// TIA Portal V20 export
// export: Created 2025-12-01T14:57:05.1586279Z, ExportSetting None, DisplayName Totally Integrated Automation Portal, DisplayVersion V20 Update 3, DisplayName TIA Portal Openness, DisplayVersion V20 Update 3, DisplayName TIA Portal Version Control Interface, DisplayVersion V20 Update 3, DisplayName STEP 7 Professional, DisplayVersion V20 Update 3, DisplayName STEP 7 Safety, DisplayVersion V20 Update 2, DisplayName WinCC Basic/Comfort/Advanced, DisplayVersion V20 Update 3, DisplayName WinCC Professional, DisplayVersion V20 Update 3, DisplayName WinCC Unified, DisplayVersion V20 Update 3
FUNCTION "FC806_JDT01Borrado" : Void   // FC806, LAD
TITLE = "BorrodoTracking" - Borrado de toda la Base de Datos
{ S7_Optimized_Access := 'FALSE' }
AUTHOR : TRACKING
NAME : 20130301
VERSION : 3.0
// - Borrado de todos los DB's
// - Inicializadcion del DB de DatosUT
// stored: AutoNumber false, SetENOAutomatically false
   VAR_TEMP
      NumeroUT : UInt;
      NumDB : Word;
      UTVacia : UInt;
   END_VAR
BEGIN

NETWORK
TITLE = Borrado de todos los DB's
// -------------------------------------------------------------------------------
// --- Mirar si hay que resetear
      AN    "DB801_JDT01StatusCOM".ResetBD;
      JC    _END;

// -------------------------------------------------------------------------------
// Borrado de los DB de Recepcion de Eventos

      CALL  "FC898_BorrarMensaje"
      ( DB_A_RESET := "DB802_JDT01RecepMensaje"
      );
      CALL  "FC898_BorrarMensaje"
      ( DB_A_RESET := "DB804_JDT01UltimoRecibido"
      );
      CALL  "FC898_BorrarMensaje"
      ( DB_A_RESET := "DB807_JDT01EventosRecibidos"
      );

// -------------------------------------------------------------------------------
// Borrado de los DB de Emision de Eventos

      CALL  "FC898_BorrarMensaje"
      ( DB_A_RESET := "DB803_JDT01EmisionMensaje"
      );
      CALL  "FC898_BorrarMensaje"
      ( DB_A_RESET := "DB805_JDT01UltimoEnviado"
      );
      CALL  "FC898_BorrarMensaje"
      ( DB_A_RESET := "DB806_JDT01EmisionAK"
      );
      CALL  "FC898_BorrarMensaje"
      ( DB_A_RESET := "DB808_JDT01EventosGenerados"
      );

// -------------------------------------------------------------------------------
// Borrado de los DB de la BD de Mesas
// El DB de CrucesMesas no se borra, esto es fijo para cada instalación

      CALL  "FC898_BorrarMensaje"
      ( DB_A_RESET := "DB810_ColasMesas"
      );
      CALL  "FC898_BorrarMensaje"
      ( DB_A_RESET := "DB811_ColasMckeys"
      );

      CALL  "FC898_BorrarMensaje"
      ( DB_A_RESET := "DB812_UTs_Control"
      );
      CALL  "FC898_BorrarMensaje"
      ( DB_A_RESET := "DB813_UTs_Ruta"
      );

      CALL  "FC898_BorrarMensaje"
      ( DB_A_RESET := "DB814_UTs_Etiqueta"
      );
      CALL  "FC898_BorrarMensaje"
      ( DB_A_RESET := "DB815_UTs_Datos"
      );
      CALL  "FC898_BorrarMensaje"
      ( DB_A_RESET := "DB816_UTs_TextoPantalla"
      );
      CALL  "FC898_BorrarMensaje"
      ( DB_A_RESET := "DB820_UTs_DatosQUBIQA"
      );
      CALL  "FC898_BorrarMensaje"
      ( DB_A_RESET := "DB821_UTs_DatosIKPAL"
      );


// -------------------------------------------------------------------------------
// Borrado de los DB de la BD de Dispositivos

      CALL  "FC898_BorrarMensaje"
      ( DB_A_RESET := "DB830_Dispositivos"
      );
      CALL  "FC898_BorrarMensaje"
      ( DB_A_RESET := "DB831_Mesas"
      );
      CALL  "FC898_BorrarMensaje"
      ( DB_A_RESET := "DB832_Maquinas"
      );


// -------------------------------------------------------------------------------
// Borrado de los DB Emision y Recepcion con la instalación

      CALL  "FC898_BorrarMensaje"
      ( DB_A_RESET := "DB840_Emision"
      );
      CALL  "FC898_BorrarMensaje"
      ( DB_A_RESET := "DB841_Recepcion"
      );
      CALL  "FC898_BorrarMensaje"
      ( DB_A_RESET := "DB843_RecepcionPantalla"
      );

      SET;
      R     "DB801_JDT01StatusCOM".ResetBD;
      JU    _FIN;  // El siguiente segmento no se realiza


NETWORK
TITLE = Final
// Se acabo la inicializacion
_END: L     0;
      LAR1;

// -------------------------------------------------------------------------------
// Borrado de los DB de Recepcion de Eventos, si es necesario

      OPN   "DB802_JDT01RecepMensaje";
      L     DBB [AR1, P#0.0];
      L     ' ';
      <>I;
      JC    S_31;
      CALL  "FC898_BorrarMensaje"
      ( DB_A_RESET := "DB802_JDT01RecepMensaje"
      );

S_31: OPN   "DB804_JDT01UltimoRecibido";
      L     DBB [AR1, P#0.0];
      L     ' ';
      <>I;
      JC    S_32;
      CALL  "FC898_BorrarMensaje"
      ( DB_A_RESET := "DB804_JDT01UltimoRecibido"
      );

S_32: OPN   "DB807_JDT01EventosRecibidos";
      L     DBB [AR1, P#0.0];

      L     ' ';
      <>I;
      JC    S_33;
      CALL  "FC898_BorrarMensaje"
      ( DB_A_RESET := "DB807_JDT01EventosRecibidos"
      );

// -------------------------------------------------------------------------------
// Borrado de los DB de Emision de Eventos, si es necesario

S_33: OPN   "DB803_JDT01EmisionMensaje";
      L     DBB [AR1, P#0.0];
      L     ' ';
      <>I;
      JC    S_34;
      CALL  "FC898_BorrarMensaje"
      ( DB_A_RESET := "DB803_JDT01EmisionMensaje"
      );

S_34: OPN   "DB805_JDT01UltimoEnviado";
      L     DBB [AR1, P#0.0];
      L     ' ';
      <>I;
      JC    S_35;
      CALL  "FC898_BorrarMensaje"
      ( DB_A_RESET := "DB805_JDT01UltimoEnviado"
      );

S_35: OPN   "DB806_JDT01EmisionAK";
      L     DBB [AR1, P#0.0];
      L     ' ';
      <>I;
      JC    S_36;
      CALL  "FC898_BorrarMensaje"
      ( DB_A_RESET := "DB806_JDT01EmisionAK"
      );

S_36: OPN   "DB808_JDT01EventosGenerados";
      L     DBB [AR1, P#0.0];
      L     ' ';
      <>I;
      JC    _FIN;
      CALL  "FC898_BorrarMensaje"
      ( DB_A_RESET := "DB808_JDT01EventosGenerados"
      );

_FIN: NOP   0;


END_FUNCTION
